INTERFACE I_Sensor

PROPERTY IsActive : Bool
GET
END_GET
END_PROPERTY

PROPERTY isNotActive : bool
GET
END_GET
END_PROPERTY

END_INTERFACE

(* stored: Version 1.1.0.1, ProductVersion 3.1.4024.11
   Itf I_Sensor: Id {ca1a4e12-fd40-4ca3-bc62-bedcec463099}
   Property IsActive: Id {289d611a-e3bd-4950-80b7-6cc340ac853f}
   Get Get: Id {8675194d-fa20-458f-83d8-1fbfacf02ae7}
   Property isNotActive: Id {08db8d1b-c3cc-478e-a5df-200f4936ad05}
   Get Get: Id {90cc890f-dcfc-4cfe-9ace-938a64a2681d} *)
